// LS Electric XG5000 project: 8_28
// PLC LSPLC
// module base 0 slot 0: 입출력 모듈:XBC-DR14E (DC 24V 입력 8점, 릴레이 출력 6점)

PROGRAM NewProgram (task: 스캔 프로그램)

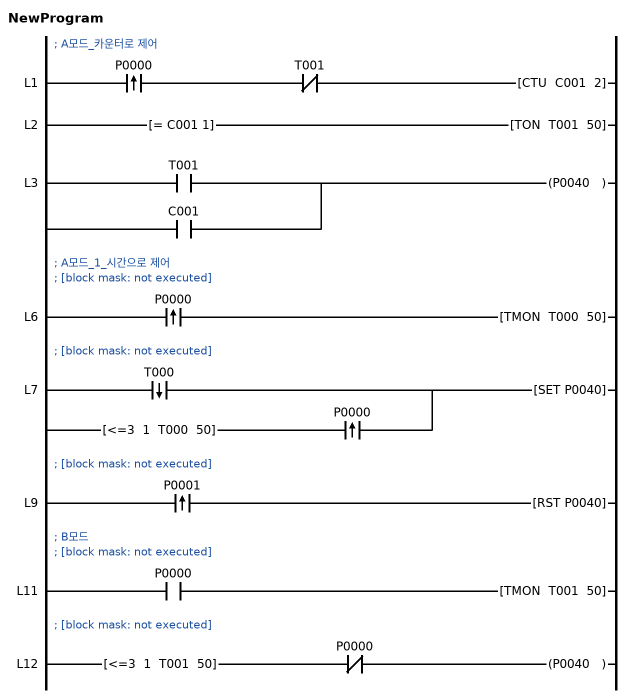
// A모드_카운터로 제어
; L1
LOADP     P0000
AND NOT   T001
CTU       C001 2
; L2
LOAD=     C001 1
TON       T001 50
; L3
LOAD      T001
OR        C001
OUT       P0040
// A모드_1_시간으로 제어
; L6 (block mask: not executed)
LOADP     P0000
TMON      T000 50
; L7 (block mask: not executed)
LOADN     T000
LOAD<=3   1 T000 50
ANDP      P0000
OR LOAD
SET       P0040
; L9 (block mask: not executed)
LOADP     P0001
RST       P0040
// B모드
; L11 (block mask: not executed)
LOAD      P0000
TMON      T001 50
; L12 (block mask: not executed)
LOAD<=3   1 T001 50
AND NOT   P0000
OUT       P0040